// TwinCAT 3 PLC project TwinCAT_OpenFramework_Devices_IO
// Title: TwinCAT Open Framework Devices IO
// Company: Oleksandr Tiutyk FOP
// Author: Oleksandr Tiutyk
// ProjectVersion: 1.0.13.0
// Description: IO devices implementation
// ProgramVersion: 3.1.4026.28
// libraries:
//   Tc2_System, * (Beckhoff Automation GmbH)
//   [TwinCAT Open Framework Automation], * (Oleksandr Tiutyk FOP)
//   [TwinCAT Open Framework Core], * (Oleksandr Tiutyk FOP)
//   [TwinCAT Open Framework IO Models], * (Oleksandr Tiutyk FOP)
// project tree:
//   Analog/Inputs/ IAnalogInputStatusProvider.TcIO, IReadOnlyAnalogInput.TcIO, AnalogInput.TcPOU (not stored), ANALOG_INPUT_STATUS.TcPOU, IAnalogInput.TcIO
//   Analog/Outputs/ IReadOnlyAnalogOutput.TcIO, AnalogOutput.TcPOU, IAnalogOutput.TcIO
//   Analog/ RawAnalogValues.TcPOU, RAW_ANALOG_VALUE.TcDUT, IAnalogValueConverter.TcIO, RAW_ANALOG_VALUE_TYPE.TcDUT
//   Analog/StandardConverters/ DirectAnalogValueConverter.TcPOU
//   Analog/StandardConverters/Range/ AbstractRangeAnalogValueConverter.TcPOU, DynamicRangeAnalogValueConverter.TcPOU, StaticRangeAnalogValueConverter.TcPOU
//   / CONTACT_TYPE.TcDUT
//   Digital/Input/ DigitalInput.TcPOU, IDigitalInput.TcIO, IReadOnlyDigitalInput.TcIO
//   Digital/Output/ DigitalOutput.TcPOU, IReadOnlyDigitalOutput.TcIO, IDigitalOutput.TcIO
//   Internal/ CurrentNamespace.TcPOU, NamespaceExtractor.TcPOU
//   Version/ Global_Version.TcGVL
// (motion and I/O tree: see PLC project twincat_openframework_core)
// real-time tasks:
//   TASK PlcTask: cycle T#10ms, priority 20, ADS port 350
//   TASK TestTask: cycle T#10ms, priority 1, ADS port 351
//   TASK RunnerTestTask: cycle T#10ms, priority 2, ADS port 354
//   TASK HowToTask: cycle T#10ms, priority 22, ADS port 353
// variable links:

// ---- Analog/RAW_ANALOG_VALUE.TcDUT
(*
SPDX-FileCopyrightText: Â© 2026 Oleksandr Tiutyk <trofimich@gmail.com>
SPDX-License-Identifier: MIT
License: https://opensource.org/license/mit
*)

(*!
<summary>4-byte union representing raw analog process data.</summary>
<description>
Allows interpreting a 4-byte raw analog signal as signed 16-bit integer, signed 32-bit integer,
or single-precision 32-bit floating point.
</description>
*)

TYPE RAW_ANALOG_VALUE :
UNION
	Int16 : INT;
	Int32 : DINT;
	Real32 : REAL; 
END_UNION
END_TYPE

// ---- Analog/RAW_ANALOG_VALUE_TYPE.TcDUT
(*
SPDX-FileCopyrightText: Â© 2026 Oleksandr Tiutyk <trofimich@gmail.com>
SPDX-License-Identifier: MIT
License: https://opensource.org/license/mit
*)

(*!
<summary>Identifies underlying data type of a raw ADC or DAC analog signal.</summary>
<description>
Specifies whether the raw process data is interpreted as signed 16-bit integer, signed 32-bit integer,
or 32-bit single-precision floating point.
</description>
*)

{attribute 'qualified_only'}
{attribute 'strict'}
{attribute 'to_string'}
TYPE RAW_ANALOG_VALUE_TYPE :
(
	INT16,
	INT32,
	REAL32 
);
END_TYPE

// ---- CONTACT_TYPE.TcDUT
(*
SPDX-FileCopyrightText: © 2026 Oleksandr Tiutyk <trofimich@gmail.com>
SPDX-License-Identifier: MIT
License: https://opensource.org/license/mit
*)

(*!
<summary>Defines electrical contact type for digital input and output signals.</summary>
<description>
Determines whether the physical signal state is inverted when mapped to the logical component Value.
NORMALLY_OPEN: logical TRUE matches physical TRUE. NORMALLY_CLOSED: logical TRUE matches physical FALSE
(inverted).
</description>
*)

{attribute 'qualified_only'}
{attribute 'strict'}
{attribute 'to_string'}
TYPE CONTACT_TYPE :
(
	NORMALLY_OPEN := 0,
	NORMALLY_CLOSED := 1
);
END_TYPE

// ---- Version/Global_Version.TcGVL
{attribute 'TcGenerated'}
{attribute 'no-analysis'}
{attribute 'linkalways'}
// This function has been automatically generated from the project information.
VAR_GLOBAL CONSTANT
	{attribute 'const_non_replaced'}
	stLibVersion_TwinCAT_Open_Framework_Devices_IO : ST_LibVersion := (iMajor := 1, iMinor := 0, iBuild := 13, iRevision := 0, nFlags := 0, sVersion := '1.0.13.0');
END_VAR

// ---- Analog/Inputs/IAnalogInputStatusProvider.TcIO
(*
SPDX-FileCopyrightText: © 2026 Oleksandr Tiutyk <trofimich@gmail.com>
SPDX-License-Identifier: MIT
License: https://opensource.org/license/mit
*)

(*!
<summary>Exposes the sampled analog input channel status by value.</summary>
<description>
A consumer of IReadOnlyAnalogInput can query this separate interface when the input supports snapshots.
</description>
*)
INTERFACE IAnalogInputStatusProvider EXTENDS TOF_Core.IObject

(*!
<summary>Gets a copy of the channel status word sampled by ProcessInput().</summary>
<description>
Returns zero before the first sample and after processing input without a status binding. Read this value
from the input's owner task. Callers can freely modify their local copy.
</description>
*)
{attribute 'monitoring' := 'call'}
PROPERTY StatusWord : WORD
GET
END_GET
END_PROPERTY

END_INTERFACE

// ---- Analog/Inputs/IReadOnlyAnalogInput.TcIO
(*
SPDX-FileCopyrightText: Â© 2026 Oleksandr Tiutyk <trofimich@gmail.com>
SPDX-License-Identifier: MIT
License: https://opensource.org/license/mit
*)

(*!
<summary>Read-only contract for an analog input component.</summary>
<description>
Provides access to engineering value, raw converter, raw ADC value, legacy decoded status, and I/O binding.
Query IAnalogInputStatusProvider for the sampled status word by value when the implementation supports it.
</description>
*)
INTERFACE IReadOnlyAnalogInput EXTENDS TOF_Automation.IInputLeafAutomationComponent,
	TOF_Core.IIOBindable

(*!
<summary>Gets the assigned analog value converter.</summary>
*)
{attribute 'monitoring' := 'call'}
PROPERTY Converter : IAnalogValueConverter
GET
END_GET
END_PROPERTY

(*!
<summary>Gets current raw hardware ADC value cast to LREAL.</summary>
*)
{attribute 'monitoring' := 'call'}
PROPERTY RawValue : LREAL
GET
END_GET
END_PROPERTY

(*!
<summary>Gets the raw analog data representation type.</summary>
*)
{attribute 'monitoring' := 'call'}
PROPERTY RawValueType : RAW_ANALOG_VALUE_TYPE
GET
END_GET
END_PROPERTY

(*!
<summary>Gets a borrowed reference to the legacy decoded channel status.</summary>
<description>
The reference requires a live input and exposes a mutable decoder. AnalogInput refreshes this view in
ProcessInput() and uses a separate sampled word for diagnostics. Use IAnalogInputStatusProvider.StatusWord
when the implementation supports reading the sampled status by value.
</description>
*)
{attribute 'monitoring' := 'call'}
PROPERTY Status : REFERENCE TO ANALOG_INPUT_STATUS
GET
END_GET
END_PROPERTY

(*!
<summary>Gets current scaled engineering unit value.</summary>
*)
{attribute 'monitoring' := 'call'}
PROPERTY Value : LREAL
GET
END_GET
END_PROPERTY

END_INTERFACE

// ---- Analog/Outputs/IReadOnlyAnalogOutput.TcIO
(*
SPDX-FileCopyrightText: Â© 2026 Oleksandr Tiutyk <trofimich@gmail.com>
SPDX-License-Identifier: MIT
License: https://opensource.org/license/mit
*)

(*!
<summary>Read-only contract for an analog output automation component.</summary>
<description>
Provides access to engineering output value, assigned converter and raw representation.
</description>
*)

INTERFACE IReadOnlyAnalogOutput EXTENDS TOF_Automation.IOutputLeafAutomationComponent

(*!
<summary>Gets the assigned analog value converter.</summary>
*)
{attribute 'monitoring' := 'call'}
PROPERTY Converter : IAnalogValueConverter
GET
END_GET
END_PROPERTY

(*!
<summary>Gets current raw hardware DAC value cast to LREAL.</summary>
*)
{attribute 'monitoring' := 'call'}
PROPERTY RawValue : LREAL
GET
END_GET
END_PROPERTY

(*!
<summary>Gets the raw analog data representation type.</summary>
*)
{attribute 'monitoring' := 'call'}
PROPERTY RawValueType : RAW_ANALOG_VALUE_TYPE
GET
END_GET
END_PROPERTY

(*!
<summary>Gets current scaled engineering unit output value.</summary>
*)
{attribute 'monitoring' := 'call'}
PROPERTY Value : LREAL
GET
END_GET
END_PROPERTY

END_INTERFACE

// ---- Analog/IAnalogValueConverter.TcIO
(*
SPDX-FileCopyrightText: Â© 2026 Oleksandr Tiutyk <trofimich@gmail.com>
SPDX-License-Identifier: MIT
License: https://opensource.org/license/mit
*)

(*!
<summary>Contract for analog signal scaling and engineering unit conversion.</summary>
<description>
Converts raw ADC/DAC values to and from engineering unit LREAL representations.
</description>
*)

INTERFACE IAnalogValueConverter EXTENDS TOF_Core.IObject

(*!
<summary>Converts an engineering unit value to raw hardware representation.</summary>
<param name="analogValue">Engineering unit analog value.</param>
<param name="rawValueType">Target raw data representation.</param>
*)
METHOD ConvertAnalogValueToRawValue : RAW_ANALOG_VALUE
VAR_INPUT
	analogValue : LREAL;
	rawValueType : RAW_ANALOG_VALUE_TYPE;
END_VAR
END_METHOD

(*!
<summary>Converts raw hardware representation to an engineering unit value.</summary>
<param name="rawValue">Raw process value union.</param>
<param name="rawValueType">Source raw data representation.</param>
*)
METHOD ConvertRawValueToAnalogValue : LREAL
VAR_INPUT
	rawValue : RAW_ANALOG_VALUE;
	rawValueType : RAW_ANALOG_VALUE_TYPE;
END_VAR
END_METHOD

END_INTERFACE

// ---- Analog/Inputs/IAnalogInput.TcIO
(*
SPDX-FileCopyrightText: Â© 2026 Oleksandr Tiutyk <trofimich@gmail.com>
SPDX-License-Identifier: MIT
License: https://opensource.org/license/mit
*)

(*!
<summary>Contract for an analog input component with channel and scalar binding capabilities.</summary>
<description>
Extends IReadOnlyAnalogInput with hardware binding methods for compound Beckhoff channels
or standalone scalar input variables.
</description>
*)
INTERFACE IAnalogInput EXTENDS IReadOnlyAnalogInput

(*!
<summary>Binds component to a 16-bit analog input channel process image structure.</summary>
<description>
Borrows the channel fields without modifying the process image. The caller keeps the channel alive while bound
and synchronizes rebinding with input processing. An invalid reference clears value and status bindings.
</description>
<param name="rawValues">Reference to channel process structure containing Status and INT Value.</param>
*)
METHOD BindToInt16IO
VAR_INPUT
	rawValues : REFERENCE TO TOF_IOModels.ANALOG_INPUT_INT_CHANNEL;
END_VAR
END_METHOD

(*!
<summary>Binds component directly to a 16-bit signed integer raw input value.</summary>
<param name="rawValue">Reference to raw INT input variable.</param>
*)
METHOD BindToInt16Value
VAR_INPUT
	rawValue : REFERENCE TO INT;
END_VAR
END_METHOD

(*!
<summary>Binds component to a 32-bit analog input channel process image structure.</summary>
<description>
Borrows the channel fields without modifying source data. The caller keeps storage alive while bound
and synchronizes rebinding with processing. An invalid reference clears value and status bindings.
The channel must use the status-plus-DINT PDO; no compact-layout or unit conversion is performed here.
</description>
<param name="rawValues">Reference to channel process structure containing Status and DINT Value.</param>
*)
METHOD BindToInt32IO
VAR_INPUT
	rawValues : REFERENCE TO TOF_IOModels.ANALOG_INPUT_DINT_CHANNEL;
END_VAR
END_METHOD

(*!
<summary>Binds component directly to a 32-bit signed integer raw input value.</summary>
<param name="rawValue">Reference to raw DINT input variable.</param>
*)
METHOD BindToInt32Value
VAR_INPUT
	rawValue : REFERENCE TO DINT;
END_VAR
END_METHOD

(*!
<summary>Binds component to a 32-bit float analog input channel process image structure.</summary>
<description>
Borrows the channel fields without modifying source data. The caller keeps storage alive while bound
and synchronizes rebinding with processing. An invalid reference clears value and status bindings.
The channel must use the status-plus-REAL PDO; no integer-layout or unit conversion is performed here.
</description>
<param name="rawValues">Reference to channel process structure containing Status and REAL Value.</param>
*)
METHOD BindToReal32IO
VAR_INPUT
	rawValues : REFERENCE TO TOF_IOModels.ANALOG_INPUT_REAL_CHANNEL;
END_VAR
END_METHOD

(*!
<summary>Binds component directly to a 32-bit single-precision float raw input value.</summary>
<param name="rawValue">Reference to raw REAL input variable.</param>
*)
METHOD BindToReal32Value
VAR_INPUT
	rawValue : REFERENCE TO REAL;
END_VAR
END_METHOD

END_INTERFACE

// ---- Analog/Outputs/IAnalogOutput.TcIO
(*
SPDX-FileCopyrightText: Â© 2026 Oleksandr Tiutyk <trofimich@gmail.com>
SPDX-License-Identifier: MIT
License: https://opensource.org/license/mit
*)

(*!
<summary>Configuration and control contract for an analog output component.</summary>
<description>
Extends IReadOnlyAnalogOutput with hardware IO binding methods and value mutator.
</description>
*)

INTERFACE IAnalogOutput EXTENDS IReadOnlyAnalogOutput

(*!
<summary>Binds component to a 16-bit signed integer output process image variable '%Q*'.</summary>
<param name="rawVariable">Reference to physical INT output variable.</param>
*)
METHOD BindToInt16IO
VAR_INPUT
	rawVariable : REFERENCE TO INT;
END_VAR
END_METHOD

(*!
<summary>Binds component to a 32-bit signed integer output process image variable '%Q*'.</summary>
<param name="rawVariable">Reference to physical DINT output variable.</param>
*)
METHOD BindToInt32IO
VAR_INPUT
	rawVariable : REFERENCE TO DINT;
END_VAR
END_METHOD

(*!
<summary>Binds component to a 32-bit float output process image variable '%Q*'.</summary>
<param name="rawVariable">Reference to physical REAL output variable.</param>
*)
METHOD BindToReal32IO
VAR_INPUT
	rawVariable : REFERENCE TO REAL;
END_VAR
END_METHOD

(*!
<summary>Gets or sets engineering unit value to output.</summary>
*)
{attribute 'monitoring' := 'call'}
PROPERTY Value : LREAL
GET
END_GET
SET
END_SET
END_PROPERTY

END_INTERFACE

// ---- Digital/Input/IDigitalInput.TcIO
(*
SPDX-FileCopyrightText: Â© 2026 Oleksandr Tiutyk <trofimich@gmail.com>
SPDX-License-Identifier: MIT
License: https://opensource.org/license/mit
*)

(*!
<summary>Configuration and binding contract for a digital input component.</summary>
<description>
Extends IReadOnlyDigitalInput with hardware IO mapping and contact type mutator.
</description>
*)

INTERFACE IDigitalInput EXTENDS IReadOnlyDigitalInput

(*!
<summary>Binds the component to a raw boolean process image variable.</summary>
<param name="rawValue">Reference to physical boolean input variable '%I*'.</param>
*)
METHOD BindToIO
VAR_INPUT
	rawValue : REFERENCE TO BOOL;
END_VAR
END_METHOD

(*!
<summary>Gets or sets electrical contact configuration.</summary>
*)
{attribute 'monitoring' := 'call'}
PROPERTY ContactType : CONTACT_TYPE
GET
END_GET
SET
END_SET
END_PROPERTY

END_INTERFACE

// ---- Digital/Input/IReadOnlyDigitalInput.TcIO
(*
SPDX-FileCopyrightText: Â© 2026 Oleksandr Tiutyk <trofimich@gmail.com>
SPDX-License-Identifier: MIT
License: https://opensource.org/license/mit
*)

(*!
<summary>Read-only contract for a digital input automation component.</summary>
<description>
Provides access to logical boolean state, change detection and electrical contact configuration.
</description>
*)

INTERFACE IReadOnlyDigitalInput EXTENDS TOF_Automation.IInputLeafAutomationComponent

(*!
<summary>Indicates whether the logical Value has changed compared to the previous cycle.</summary>
*)
{attribute 'monitoring' := 'call'}
PROPERTY Changed : BOOL
GET
END_GET
END_PROPERTY

(*!
<summary>Gets electrical contact configuration (normally open or normally closed).</summary>
*)
{attribute 'monitoring' := 'call'}
PROPERTY ContactType : CONTACT_TYPE
GET
END_GET
END_PROPERTY

(*!
<summary>Gets current evaluated logical state of the input signal.</summary>
*)
{attribute 'monitoring' := 'call'}
PROPERTY Value : BOOL
GET
END_GET
END_PROPERTY

END_INTERFACE

// ---- Digital/Output/IReadOnlyDigitalOutput.TcIO
(*
SPDX-FileCopyrightText: Â© 2026 Oleksandr Tiutyk <trofimich@gmail.com>
SPDX-License-Identifier: MIT
License: https://opensource.org/license/mit
*)

(*!
<summary>Read-only contract for a digital output automation component.</summary>
<description>
Provides access to logical boolean output state, change detection and electrical contact configuration.
</description>
*)

INTERFACE IReadOnlyDigitalOutput EXTENDS TOF_Automation.IOutputLeafAutomationComponent

(*!
<summary>Indicates whether the current logical command differs from the last processed command.</summary>
<description>
ProcessOutput() acknowledges the current command even without an I/O binding.
</description>
*)
{attribute 'monitoring' := 'call'}
PROPERTY Changed : BOOL
GET
END_GET
END_PROPERTY

(*!
<summary>Gets electrical contact configuration.</summary>
*)
{attribute 'monitoring' := 'call'}
PROPERTY ContactType : CONTACT_TYPE
GET
END_GET
END_PROPERTY

(*!
<summary>Gets current evaluated logical state of the output signal.</summary>
*)
{attribute 'monitoring' := 'call'}
PROPERTY Value : BOOL
GET
END_GET
END_PROPERTY

END_INTERFACE

// ---- Digital/Output/IDigitalOutput.TcIO
(*
SPDX-FileCopyrightText: Â© 2026 Oleksandr Tiutyk <trofimich@gmail.com>
SPDX-License-Identifier: MIT
License: https://opensource.org/license/mit
*)

(*!
<summary>Configuration and control contract for a digital output component.</summary>
<description>
Extends IReadOnlyDigitalOutput with hardware IO mapping, contact configuration and state setter.
</description>
*)

INTERFACE IDigitalOutput EXTENDS IReadOnlyDigitalOutput

(*!
<summary>Binds component to a raw boolean process image output variable.</summary>
<param name="rawValue">Reference to physical boolean output variable '%Q*'.</param>
*)
METHOD BindToIO
VAR_INPUT
	rawValue : REFERENCE TO BOOL;
END_VAR
END_METHOD

(*!
<summary>Gets or sets electrical contact configuration.</summary>
*)
{attribute 'monitoring' := 'call'}
PROPERTY ContactType : CONTACT_TYPE
GET
END_GET
SET
END_SET
END_PROPERTY

(*!
<summary>Gets or sets logical state to write to the digital output.</summary>
*)
{attribute 'monitoring' := 'call'}
PROPERTY Value : BOOL
GET
END_GET
SET
END_SET
END_PROPERTY

END_INTERFACE

// ---- Analog/RawAnalogValues.TcPOU
(*
SPDX-FileCopyrightText: Â© 2026 Oleksandr Tiutyk <trofimich@gmail.com>
SPDX-License-Identifier: MIT
License: https://opensource.org/license/mit
*)

(*!
<summary>Utility program providing factory methods to construct RAW_ANALOG_VALUE unions.</summary>
<description>
Ensures that unused bytes of the 4-byte union are zero-initialized when constructing from 16-bit values.
</description>
*)

{attribute 'no_explicit_call' := 'do not call this POU directly'}
PROGRAM RawAnalogValues
VAR
	{attribute 'hide'} 
	_ClassName : STRING := __POUNAME();
END_VAR

(*!
<summary>Gets the class name of the program.</summary>
*)
{attribute 'monitoring' := 'call'}
PROPERTY ClassName : REFERENCE TO STRING
GET
ClassName REF= _ClassName;
END_GET
END_PROPERTY

(*!
<summary>Creates a RAW_ANALOG_VALUE union from a 16-bit signed integer.</summary>
<description>Zeroes upper bytes of the 4-byte union before assigning the 16-bit value.</description>
<param name="value">16-bit signed integer value.</param>
*)
METHOD FromInt16 : RAW_ANALOG_VALUE
VAR_INPUT
	value : INT;
END_VAR
FromInt16.Int32 := 0;
FromInt16.Int16 := value;
END_METHOD

(*!
<summary>Creates a RAW_ANALOG_VALUE union from a 32-bit signed integer.</summary>
<param name="value">32-bit signed integer value.</param>
*)
METHOD FromInt32 : RAW_ANALOG_VALUE
VAR_INPUT
	value : DINT;
END_VAR
FromInt32.Int32 := value;
END_METHOD

(*!
<summary>Creates a RAW_ANALOG_VALUE union from a 32-bit single-precision float.</summary>
<param name="value">32-bit float value.</param>
*)
METHOD FromReal32 : RAW_ANALOG_VALUE
VAR_INPUT
	value : REAL;
END_VAR
FromReal32.Real32 := value;
END_METHOD

(*!
<summary>Gets the namespace name of the program.</summary>
*)
{attribute 'monitoring' := 'call'}
PROPERTY NamespaceName : REFERENCE TO STRING
GET
NamespaceName REF= CurrentNamespace.Name;
END_GET
END_PROPERTY

END_PROGRAM

// ---- Internal/CurrentNamespace.TcPOU
(*
SPDX-FileCopyrightText: Â© 2026 Oleksandr Tiutyk <trofimich@gmail.com>
SPDX-License-Identifier: MIT
License: https://opensource.org/license/mit
*)

(*!
<summary>Internal program providing library namespace extraction.</summary>
*)

{attribute 'no_explicit_call' := 'do not call this POU directly'}
PROGRAM INTERNAL CurrentNamespace
VAR
	{attribute 'hide'} 
	_NamespaceExtractor : NamespaceExtractor;
END_VAR

(*!
<summary>Gets the effective namespace of this library.</summary>
*)
{attribute 'monitoring' := 'call'}
PROPERTY Name : REFERENCE TO STRING
GET
Name REF= _NamespaceExtractor.CurrentNamespace;
END_GET
END_PROPERTY

END_PROGRAM

// ---- Internal/NamespaceExtractor.TcPOU
(*
SPDX-FileCopyrightText: Â© 2026 Oleksandr Tiutyk <trofimich@gmail.com>
SPDX-License-Identifier: MIT
License: https://opensource.org/license/mit
*)

(*!
<summary>Internal function block that extracts the library namespace via init_namespace attribute.</summary>
*)

FUNCTION_BLOCK INTERNAL NamespaceExtractor
VAR_OUTPUT
	{attribute 'init_namespace'} 
	CurrentNamespace : STRING; 	
END_VAR

END_FUNCTION_BLOCK

// ---- Analog/Inputs/ANALOG_INPUT_STATUS.TcPOU
(*
SPDX-FileCopyrightText: Â© 2026 Oleksandr Tiutyk <trofimich@gmail.com>
SPDX-License-Identifier: MIT
License: https://opensource.org/license/mit
*)

(*!
<summary>Encapsulates and decodes Beckhoff 16-bit EtherCAT analog input status word.</summary>
<description>
Provides decoded boolean properties for Underrange (bit 0), Overrange (bit 1), Limit 1 (bits 2..3),
Limit 2 (bits 4..5), Error (bit 6), TxPDO State (bit 14), and TxPDO Toggle (bit 15).
</description>
*)

FUNCTION_BLOCK ANALOG_INPUT_STATUS
VAR
	_Status : WORD;
END_VAR

(*!
<summary>Bit 6: General measurement or hardware error flag.</summary>
*)
{attribute 'monitoring' := 'call'}
PROPERTY FINAL Error : BOOL
GET
Error := _Status.6;
END_GET
END_PROPERTY

(*!
<summary>Bit 1: Upper limit of nominal measuring range exceeded.</summary>
*)
{attribute 'monitoring' := 'call'}
PROPERTY FINAL Overrange : BOOL
GET
Overrange := _Status.1;
END_GET
END_PROPERTY

(*!
<summary>Updates internal raw 16-bit status word.</summary>
<param name="status">Raw 16-bit EtherCAT channel status word.</param>
*)
METHOD SetStatus
VAR_INPUT
	status : WORD;
END_VAR
_Status := status;
END_METHOD

(*!
<summary>Bit 14: TxPDO data validity (0: valid, 1: invalid / bus error).</summary>
*)
{attribute 'monitoring' := 'call'}
PROPERTY FINAL TxPDOState : BOOL
GET
TxPDOState := _Status.14;
END_GET
END_PROPERTY

(*!
<summary>Bit 15: TxPDO communication toggle bit.</summary>
*)
{attribute 'monitoring' := 'call'}
PROPERTY FINAL TxPDOToggle : BOOL
GET
TxPDOToggle := _Status.15;
END_GET
END_PROPERTY

(*!
<summary>Bit 0: Lower limit of calibrated measuring range fallen below.</summary>
*)
{attribute 'monitoring' := 'call'}
PROPERTY FINAL Underrange : BOOL
GET
Underrange := _Status.0;
END_GET
END_PROPERTY

(*!
<summary>Bit 3: Input value is greater than or equal to Limit 1 threshold.</summary>
*)
{attribute 'monitoring' := 'call'}
PROPERTY FINAL ValueBiggerOrEqualLimit1 : BOOL
GET
ValueBiggerOrEqualLimit1 := _Status.3;
END_GET
END_PROPERTY

(*!
<summary>Bit 5: Input value is greater than or equal to Limit 2 threshold.</summary>
*)
{attribute 'monitoring' := 'call'}
PROPERTY FINAL ValueBiggerOrEqualLimit2 : BOOL
GET
ValueBiggerOrEqualLimit2 := _Status.5;
END_GET
END_PROPERTY

(*!
<summary>Bit 2: Input value is smaller than or equal to Limit 1 threshold.</summary>
*)
{attribute 'monitoring' := 'call'}
PROPERTY FINAL ValueSmallerOrEqualLimit1 : BOOL
GET
ValueSmallerOrEqualLimit1 := _Status.2;
END_GET
END_PROPERTY

(*!
<summary>Bit 4: Input value is smaller than or equal to Limit 2 threshold.</summary>
*)
{attribute 'monitoring' := 'call'}
PROPERTY FINAL ValueSmallerOrEqualLimit2 : BOOL
GET
ValueSmallerOrEqualLimit2 := _Status.4;
END_GET
END_PROPERTY

END_FUNCTION_BLOCK

// ---- Analog/Outputs/AnalogOutput.TcPOU
(*
SPDX-FileCopyrightText: Â© 2026 Oleksandr Tiutyk <trofimich@gmail.com>
SPDX-License-Identifier: MIT
License: https://opensource.org/license/mit
*)

(*!
<summary>Analog output automation component converting engineering values into raw DAC signals.</summary>
<description>
Scales engineering unit values using an assigned IAnalogValueConverter and writes raw data to hardware outputs.
Successful initialization requires a parent automation component.
</description>
*)

FUNCTION_BLOCK AnalogOutput EXTENDS TOF_Automation.OutputLeafAutomationComponent
	IMPLEMENTS IAnalogOutput, TOF_Core.IIOBindable
VAR_STAT
	{attribute 'hide'} 
	_ClassName : STRING := __POUNAME();
END_VAR
VAR	
	{attribute 'hide'} 
	_RawValueType : RAW_ANALOG_VALUE_TYPE;

	{attribute 'hide'} 
	_Converter : IAnalogValueConverter;

	_CurrentValue : LREAL;
	_PreviousValue : LREAL;
	
	_RawInt16Value : REFERENCE TO INT;
	_RawInt32Value : REFERENCE TO DINT;
	_RawReal32Value : REFERENCE TO REAL; 
END_VAR

(*!
<summary>Binds component to a 16-bit signed integer output process image variable '%Q*'.</summary>
<param name="rawVariable">Reference to physical INT output variable.</param>
*)
METHOD BindToInt16IO
VAR_INPUT
	rawVariable : REFERENCE TO INT;
END_VAR
_RawValueType := RAW_ANALOG_VALUE_TYPE.INT16;

_RawInt16Value REF= rawVariable;
_RawInt32Value REF= 0;
_RawReal32Value REF= 0;
END_METHOD

(*!
<summary>Binds component to a 32-bit signed integer output process image variable '%Q*'.</summary>
<param name="rawVariable">Reference to physical DINT output variable.</param>
*)
METHOD BindToInt32IO
VAR_INPUT
	rawVariable : REFERENCE TO DINT;
END_VAR
_RawValueType := RAW_ANALOG_VALUE_TYPE.INT32;

_RawInt16Value REF= 0;
_RawInt32Value REF= rawVariable;
_RawReal32Value REF= 0;
END_METHOD

(*!
<summary>Binds component to a 32-bit float output process image variable '%Q*'.</summary>
<param name="rawVariable">Reference to physical REAL output variable.</param>
*)
METHOD BindToReal32IO
VAR_INPUT
	rawVariable : REFERENCE TO REAL;
END_VAR
_RawValueType := RAW_ANALOG_VALUE_TYPE.REAL32;

_RawInt16Value REF= 0;
_RawInt32Value REF= 0;
_RawReal32Value REF= rawVariable;
END_METHOD

(*!
<summary>Gets whether the component raw value is bound to a valid physical IO variable.</summary>
*)
{attribute 'monitoring' := 'call'}
PROPERTY FINAL BoundToIO : BOOL
GET
CASE _RawValueType OF
	RAW_ANALOG_VALUE_TYPE.INT16:
		BoundToIO := __ISVALIDREF(_RawInt16Value);
	
	RAW_ANALOG_VALUE_TYPE.INT32:
		BoundToIO := __ISVALIDREF(_RawInt32Value);
	
	RAW_ANALOG_VALUE_TYPE.REAL32:
		BoundToIO := __ISVALIDREF(_RawReal32Value);
END_CASE
END_GET
END_PROPERTY

(*!
<summary>Gets the class name of the component.</summary>
*)
{attribute 'monitoring' := 'call'}
PROPERTY ClassName : REFERENCE TO STRING
GET
ClassName REF= _ClassName;
END_GET
END_PROPERTY

(*!
<summary>Gets the assigned analog value converter.</summary>
*)
{attribute 'monitoring' := 'call'}
PROPERTY FINAL Converter : IAnalogValueConverter
GET
Converter := _Converter;
END_GET
END_PROPERTY

(*!
<summary>Initializes component name, parent and converter dependency.</summary>
<param name="bInitRetains">TRUE: retain variables are initialized.</param>
<param name="bInCopyCode">TRUE: instance copied to copy code (online change).</param>
<param name="name">Component instance name.</param>
<param name="parent">Nonzero parent automation component required for successful Initialize().</param>
<param name="converter">Mandatory analog value converter dependency.</param>
*)
METHOD FB_init : BOOL
VAR_INPUT
	bInitRetains : BOOL; // TRUE: the retain variables are initialized (reset warm / reset cold)
	bInCopyCode : BOOL;  // TRUE: the instance will be copied to the copy code afterward (online change)
	name : WSTRING;
	parent : TOF_Automation.IParentAutomationComponent;
	converter : IAnalogValueConverter;
END_VAR
IF NOT bInCopyCode THEN
	_Converter := converter;
END_IF
END_METHOD

(*!
<summary>Gets the namespace name of the component.</summary>
*)
{attribute 'monitoring' := 'call'}
PROPERTY NamespaceName : REFERENCE TO STRING
GET
NamespaceName REF= CurrentNamespace.Name;
END_GET
END_PROPERTY

(*!
<summary>Validates that mandatory converter dependency is configured.</summary>
*)
METHOD PROTECTED OnInitializing : BOOL
IF _Converter = 0 THEN
	TOF_Core.Exceptions.ThrowClassInitialization(
		sourceNamespaceName := NamespaceName,
		sourceClassName := ClassName,
		sourcePOUName := __POUNAME(),
		sourcePosition := __POSITION(),
		errorMessage := "converter not specified"
	);
END_IF

OnInitializing := TRUE;
END_METHOD

(*!
<summary>Scales engineering value to raw DAC signal and writes to bound hardware output.</summary>
*)
METHOD PROTECTED OnProcessOutput
setRawValueByUnion(
	_Converter.ConvertAnalogValueToRawValue(
		analogValue := _CurrentValue,
		rawValueType := _RawValueType
	)
);

_PreviousValue := _CurrentValue;
END_METHOD

(*!
<summary>Gets current raw hardware DAC value cast to LREAL.</summary>
*)
{attribute 'monitoring' := 'call'}
PROPERTY FINAL RawValue : LREAL
GET
CASE _RawValueType OF
	RAW_ANALOG_VALUE_TYPE.INT16:
		RawValue := SEL(__ISVALIDREF(_RawInt16Value), 0, TO_LREAL(_RawInt16Value));
	
	RAW_ANALOG_VALUE_TYPE.INT32:
		RawValue := SEL(__ISVALIDREF(_RawInt32Value), 0, TO_LREAL(_RawInt32Value));
	
	RAW_ANALOG_VALUE_TYPE.REAL32:
		RawValue := SEL(__ISVALIDREF(_RawReal32Value), 0, TO_LREAL(_RawReal32Value));
END_CASE
END_GET
END_PROPERTY

(*!
<summary>Gets the raw analog data representation type.</summary>
*)
{attribute 'monitoring' := 'call'}
PROPERTY FINAL RawValueType : RAW_ANALOG_VALUE_TYPE
GET
RawValueType := _RawValueType;
END_GET
END_PROPERTY

(*!
<summary>Gets the memory size of the instance.</summary>
*)
{attribute 'monitoring' := 'call'}
PROPERTY SelfSize : ULINT
GET
SelfSize := XSIZEOF(THIS^);
END_GET
END_PROPERTY

METHOD PRIVATE setRawValueByUnion
VAR_INPUT
	rawValueUnion : RAW_ANALOG_VALUE;
END_VAR
CASE _RawValueType OF
	RAW_ANALOG_VALUE_TYPE.INT16:
		IF __ISVALIDREF(_RawInt16Value) THEN
			_RawInt16Value := rawValueUnion.Int16; 
		END_IF
	
	RAW_ANALOG_VALUE_TYPE.INT32:
		IF __ISVALIDREF(_RawInt32Value) THEN
			_RawInt32Value := rawValueUnion.Int32; 
		END_IF
	
	RAW_ANALOG_VALUE_TYPE.REAL32:
		IF __ISVALIDREF(_RawReal32Value) THEN
			_RawReal32Value := rawValueUnion.Real32; 
		END_IF
END_CASE
END_METHOD

(*!
<summary>Gets or sets engineering unit value to output.</summary>
*)
{attribute 'monitoring' := 'call'}
PROPERTY Value : LREAL
GET
Value := _CurrentValue;
END_GET
SET
_CurrentValue := Value;
END_SET
END_PROPERTY

END_FUNCTION_BLOCK

// ---- Analog/StandardConverters/DirectAnalogValueConverter.TcPOU
(*
SPDX-FileCopyrightText: Â© 2026 Oleksandr Tiutyk <trofimich@gmail.com>
SPDX-License-Identifier: MIT
License: https://opensource.org/license/mit
*)

(*!
<summary>Performs direct 1:1 pass-through conversion between raw and engineering analog values.</summary>
<description>
Casts between numeric types without range scaling or boundary clamping.
</description>
*)

{attribute 'no_explicit_call' := 'do not call this function block directly'}
FUNCTION_BLOCK DirectAnalogValueConverter EXTENDS TOF_Core.Object IMPLEMENTS IAnalogValueConverter
VAR_STAT
	{attribute 'hide'} 
	_ClassName : STRING := __POUNAME();
END_VAR

(*!
<summary>Gets the class name of the converter.</summary>
*)
{attribute 'monitoring' := 'call'}
PROPERTY ClassName : REFERENCE TO STRING
GET
ClassName REF= _ClassName;
END_GET
END_PROPERTY

(*!
<summary>Directly converts an engineering unit value to raw hardware representation.</summary>
<param name="analogValue">Engineering unit analog value.</param>
<param name="rawValueType">Target raw data representation.</param>
*)
METHOD ConvertAnalogValueToRawValue : RAW_ANALOG_VALUE
VAR_INPUT
	analogValue	: LREAL;
	rawValueType : RAW_ANALOG_VALUE_TYPE;
END_VAR
ConvertAnalogValueToRawValue.Int32 := 0;

CASE rawValueType OF
	RAW_ANALOG_VALUE_TYPE.INT16:
		ConvertAnalogValueToRawValue.Int16 := TO_INT(analogValue);
	
	RAW_ANALOG_VALUE_TYPE.INT32:
		ConvertAnalogValueToRawValue.Int32 := TO_DINT(analogValue);
	
	RAW_ANALOG_VALUE_TYPE.REAL32:
		ConvertAnalogValueToRawValue.Real32 := TO_REAL(analogValue);
	
	ELSE
		RETURN;
END_CASE
END_METHOD

(*!
<summary>Directly converts a raw hardware representation to an engineering unit value.</summary>
<param name="rawValue">Raw process value union.</param>
<param name="rawValueType">Source raw data representation.</param>
*)
METHOD ConvertRawValueToAnalogValue : LREAL
VAR_INPUT
	rawValue : RAW_ANALOG_VALUE;
	rawValueType : RAW_ANALOG_VALUE_TYPE;
END_VAR
CASE rawValueType OF
	RAW_ANALOG_VALUE_TYPE.INT16:
		ConvertRawValueToAnalogValue := TO_LREAL(rawValue.Int16);
	
	RAW_ANALOG_VALUE_TYPE.INT32:
		ConvertRawValueToAnalogValue := TO_LREAL(rawValue.Int32);
	
	RAW_ANALOG_VALUE_TYPE.REAL32:
		ConvertRawValueToAnalogValue := TO_LREAL(rawValue.Real32);
	
	ELSE
		ConvertRawValueToAnalogValue := 0;
END_CASE
END_METHOD

(*!
<summary>Gets the namespace name of the converter.</summary>
*)
{attribute 'monitoring' := 'call'}
PROPERTY NamespaceName : REFERENCE TO STRING
GET
NamespaceName REF= CurrentNamespace.Name;
END_GET
END_PROPERTY

(*!
<summary>Gets the memory size of the instance.</summary>
*)
{attribute 'monitoring' := 'call'}
PROPERTY SelfSize : ULINT
GET
SelfSize := XSIZEOF(THIS^);
END_GET
END_PROPERTY

END_FUNCTION_BLOCK

// ---- Analog/StandardConverters/Range/AbstractRangeAnalogValueConverter.TcPOU
(*
SPDX-FileCopyrightText: Â© 2026 Oleksandr Tiutyk <trofimich@gmail.com>
SPDX-License-Identifier: MIT
License: https://opensource.org/license/mit
*)

(*!
<summary>Base converter providing linear interpolation and boundary clamping
between raw and engineering values.</summary>
<description>
Maps an input value proportionally between configured minimum and maximum limits.
Clamps values outside range to boundary limits and defends against division by zero.
For a range with distinct engineering limits and equal raw limits, output conversion returns the common raw limit.
</description>
*)

{attribute 'no_explicit_call' := 'do not call this function block directly'}
FUNCTION_BLOCK ABSTRACT AbstractRangeAnalogValueConverter EXTENDS TOF_Core.Object IMPLEMENTS IAnalogValueConverter
VAR
	{attribute 'hide'} 
	_MinAnalogValue : REFERENCE TO LREAL;
	{attribute 'hide'} 
	_MaxAnalogValue : REFERENCE TO LREAL;
	{attribute 'hide'} 
	_MinRawValue : REFERENCE TO RAW_ANALOG_VALUE;
	{attribute 'hide'} 
	_MaxRawValue : REFERENCE TO RAW_ANALOG_VALUE;
END_VAR

(*!
<summary>Converts an engineering unit value to raw hardware representation with boundary clamping.</summary>
<description>
If the engineering limits differ and the raw limits are equal, returns the common limit in the requested
raw representation. An INT16 result has zeroed upper bytes.
</description>
<param name="analogValue">Engineering unit analog value.</param>
<param name="rawValueType">Target raw data representation.</param>
*)
METHOD ConvertAnalogValueToRawValue : RAW_ANALOG_VALUE
VAR_INPUT
	analogValue	: LREAL;
	rawValueType : RAW_ANALOG_VALUE_TYPE;
END_VAR
VAR
	formattedExceptionMessage : TOF_Core.ERROR_MESSAGE;

	minRawValueLReal : LREAL;
	maxRawValueLReal : LREAL;
	rawValueLReal : LREAL;
	
	exceptionCode : __SYSTEM.ExceptionCode;	
END_VAR
IF NOT __ISVALIDREF(_MinAnalogValue)
	OR_ELSE NOT __ISVALIDREF(_MaxAnalogValue)
	OR_ELSE NOT __ISVALIDREF(_MinRawValue)
	OR_ELSE NOT __ISVALIDREF(_MaxRawValue)
	OR_ELSE _MinAnalogValue = _MaxAnalogValue
THEN
	RETURN;
END_IF

IF _MaxAnalogValue > _MinAnalogValue THEN
	IF analogValue >= _MaxAnalogValue THEN
		analogValue := _MaxAnalogValue;
	ELSIF analogValue <= _MinAnalogValue THEN
		analogValue := _MinAnalogValue;
	END_IF
ELSIF _MaxAnalogValue < _MinAnalogValue THEN
	IF analogValue <= _MaxAnalogValue THEN
		analogValue := _MaxAnalogValue;
	ELSIF analogValue >= _MinAnalogValue THEN
		analogValue := _MinAnalogValue;
	END_IF
END_IF

CASE rawValueType OF
	RAW_ANALOG_VALUE_TYPE.INT16:
		minRawValueLReal := TO_LREAL(_MinRawValue.Int16);
		maxRawValueLReal := TO_LREAL(_MaxRawValue.Int16);

	RAW_ANALOG_VALUE_TYPE.INT32:
		minRawValueLReal := TO_LREAL(_MinRawValue.Int32);
		maxRawValueLReal := TO_LREAL(_MaxRawValue.Int32);

	RAW_ANALOG_VALUE_TYPE.REAL32:
		minRawValueLReal := TO_LREAL(_MinRawValue.Real32);
		maxRawValueLReal := TO_LREAL(_MaxRawValue.Real32);

	ELSE
		RETURN;
END_CASE

IF minRawValueLReal = maxRawValueLReal THEN
	CASE rawValueType OF
		RAW_ANALOG_VALUE_TYPE.INT16:
			ConvertAnalogValueToRawValue := RawAnalogValues.FromInt16(value := _MinRawValue.Int16);

		RAW_ANALOG_VALUE_TYPE.INT32:
			ConvertAnalogValueToRawValue := RawAnalogValues.FromInt32(value := _MinRawValue.Int32);

		RAW_ANALOG_VALUE_TYPE.REAL32:
			ConvertAnalogValueToRawValue := RawAnalogValues.FromReal32(value := _MinRawValue.Real32);
	END_CASE

	RETURN;
END_IF

__TRY
	rawValueLReal := (analogValue - _MinAnalogValue) / (_MaxAnalogValue - _MinAnalogValue)
		* (maxRawValueLReal - minRawValueLReal) + minRawValueLReal;
__CATCH(exceptionCode)
	formattedExceptionMessage := TOF_Core.WideStrings.Concat255(
		"Invalid analog to raw value conversion. Exception code: ",
		TO_WSTRING(exceptionCode)
	);

	TOF_Core.Exceptions.ThrowStandard(
		sourceNamespaceName := NamespaceName,
		sourceClassName := ClassName,
		sourcePOUName := __POUNAME(),
		sourcePosition := __POSITION(),
		message := formattedExceptionMessage
	);
__ENDTRY

ConvertAnalogValueToRawValue.Int32 := 0;

CASE rawValueType OF
	RAW_ANALOG_VALUE_TYPE.INT16:
		ConvertAnalogValueToRawValue.Int16 := TO_INT(rawValueLReal);

	RAW_ANALOG_VALUE_TYPE.INT32:
		ConvertAnalogValueToRawValue.Int32 := TO_DINT(rawValueLReal);

	RAW_ANALOG_VALUE_TYPE.REAL32:
		ConvertAnalogValueToRawValue.Real32 := TO_REAL(rawValueLReal);
END_CASE
END_METHOD

(*!
<summary>Converts raw hardware representation to an engineering unit value with boundary clamping.</summary>
<param name="rawValue">Raw process value union.</param>
<param name="rawValueType">Source raw data representation.</param>
*)
METHOD ConvertRawValueToAnalogValue : LREAL
VAR_INPUT
	rawValue : RAW_ANALOG_VALUE;
	rawValueType : RAW_ANALOG_VALUE_TYPE;
END_VAR
VAR
	formattedExceptionMessage : TOF_Core.ERROR_MESSAGE;

	rawValueLReal : LREAL;
	minRawValueLReal : LREAL;
	maxRawValueLReal : LREAL;

	exceptionCode : __SYSTEM.ExceptionCode;
END_VAR
IF NOT __ISVALIDREF(_MinAnalogValue)
	OR_ELSE NOT __ISVALIDREF(_MaxAnalogValue)
	OR_ELSE NOT __ISVALIDREF(_MinRawValue)
	OR_ELSE NOT __ISVALIDREF(_MaxRawValue)
	OR_ELSE _MinAnalogValue = _MaxAnalogValue
THEN
	RETURN;
END_IF

CASE rawValueType OF
	RAW_ANALOG_VALUE_TYPE.INT16:
		rawValueLReal := TO_LREAL(rawValue.Int16);
		minRawValueLReal := TO_LREAL(_MinRawValue.Int16);
		maxRawValueLReal := TO_LREAL(_MaxRawValue.Int16);

	RAW_ANALOG_VALUE_TYPE.INT32:
		rawValueLReal := TO_LREAL(rawValue.Int32);
		minRawValueLReal := TO_LREAL(_MinRawValue.Int32);
		maxRawValueLReal := TO_LREAL(_MaxRawValue.Int32);

	RAW_ANALOG_VALUE_TYPE.REAL32:
		rawValueLReal := TO_LREAL(rawValue.Real32);
		minRawValueLReal := TO_LREAL(_MinRawValue.Real32);
		maxRawValueLReal := TO_LREAL(_MaxRawValue.Real32);

	ELSE
		RETURN;
END_CASE

IF maxRawValueLReal > minRawValueLReal THEN
	IF rawValueLReal >= maxRawValueLReal THEN
		ConvertRawValueToAnalogValue := _MaxAnalogValue;
		RETURN;
	ELSIF rawValueLReal <= minRawValueLReal THEN
		ConvertRawValueToAnalogValue := _MinAnalogValue;
		RETURN;
	END_IF
ELSIF maxRawValueLReal < minRawValueLReal THEN
	IF rawValueLReal <= maxRawValueLReal THEN
		ConvertRawValueToAnalogValue := _MaxAnalogValue;
		RETURN;
	ELSIF rawValueLReal >= minRawValueLReal THEN
		ConvertRawValueToAnalogValue := _MinAnalogValue;
		RETURN;
	END_IF
ELSE
	ConvertRawValueToAnalogValue := _MinAnalogValue;
	RETURN;
END_IF

__TRY
	ConvertRawValueToAnalogValue := (rawValueLReal - minRawValueLReal) / (maxRawValueLReal - minRawValueLReal)
		* (_MaxAnalogValue - _MinAnalogValue) + _MinAnalogValue;
__CATCH(exceptionCode)
	formattedExceptionMessage := TOF_Core.WideStrings.Concat255(
		"Invalid raw to analog value conversion. Exception code: ",
		TO_WSTRING(exceptionCode)
	);

	TOF_Core.Exceptions.ThrowStandard(
		sourceNamespaceName := NamespaceName,
		sourceClassName := ClassName,
		sourcePOUName := __POUNAME(),
		sourcePosition := __POSITION(),
		message := formattedExceptionMessage
	);
__ENDTRY
END_METHOD

(*!
<summary>Gets a reference to the maximum engineering unit value.</summary>
*)
{attribute 'monitoring' := 'call'}
PROPERTY FINAL MaxAnalogValue : REFERENCE TO LREAL
GET
MaxAnalogValue REF= _MaxAnalogValue;
END_GET
END_PROPERTY

(*!
<summary>Gets a reference to the maximum raw process value.</summary>
*)
{attribute 'monitoring' := 'call'}
PROPERTY FINAL MaxRawValue : REFERENCE TO RAW_ANALOG_VALUE
GET
MaxRawValue REF= _MaxRawValue;
END_GET
END_PROPERTY

(*!
<summary>Gets a reference to the minimum engineering unit value.</summary>
*)
{attribute 'monitoring' := 'call'}
PROPERTY FINAL MinAnalogValue : REFERENCE TO LREAL
GET
MinAnalogValue REF= _MinAnalogValue;
END_GET
END_PROPERTY

(*!
<summary>Gets a reference to the minimum raw process value.</summary>
*)
{attribute 'monitoring' := 'call'}
PROPERTY FINAL MinRawValue : REFERENCE TO RAW_ANALOG_VALUE
GET
MinRawValue REF= _MinRawValue;
END_GET
END_PROPERTY

(*!
<summary>Gets the namespace name of the converter.</summary>
*)
{attribute 'monitoring' := 'call'}
PROPERTY NamespaceName : REFERENCE TO STRING
GET
NamespaceName REF= CurrentNamespace.Name;
END_GET
END_PROPERTY

END_FUNCTION_BLOCK

// ---- Analog/StandardConverters/Range/DynamicRangeAnalogValueConverter.TcPOU
(*
SPDX-FileCopyrightText: Â© 2026 Oleksandr Tiutyk <trofimich@gmail.com>
SPDX-License-Identifier: MIT
License: https://opensource.org/license/mit
*)

(*!
<summary>Range converter with dynamically referenced limit variables that can change at runtime.</summary>
<description>
Safely handles online changes without resetting dynamic references to zero.
</description>
*)

{attribute 'no_explicit_call' := 'do not call this function block directly'}
FUNCTION_BLOCK DynamicRangeAnalogValueConverter EXTENDS AbstractRangeAnalogValueConverter
VAR_STAT
	{attribute 'hide'} 
	_ClassName : STRING := __POUNAME();
END_VAR
VAR
	{attribute 'hide'} 
	_ZeroAnalogValue : LREAL;
	{attribute 'hide'} 
	_ZeroRawValue : RAW_ANALOG_VALUE; 
END_VAR

(*!
<summary>Gets the class name of the converter.</summary>
*)
{attribute 'monitoring' := 'call'}
PROPERTY ClassName : REFERENCE TO STRING
GET
ClassName REF= _ClassName;
END_GET
END_PROPERTY

(*!
<summary>Initializes dynamic limit references.</summary>
<param name="bInitRetains">TRUE: retain variables are initialized.</param>
<param name="bInCopyCode">TRUE: instance copied to copy code (online change).</param>
<param name="minAnalogValue">Reference to minimum engineering unit variable.</param>
<param name="maxAnalogValue">Reference to maximum engineering unit variable.</param>
<param name="minRawValue">Reference to minimum raw process variable.</param>
<param name="maxRawValue">Reference to maximum raw process variable.</param>
*)
METHOD FB_init : BOOL
VAR_INPUT
	bInitRetains : BOOL; // TRUE: the retain variables are initialized (reset warm / reset cold)
	bInCopyCode : BOOL;  // TRUE: the instance will be copied to the copy code afterward (online change)
	minAnalogValue : REFERENCE TO LREAL;
	maxAnalogValue : REFERENCE TO LREAL;
	minRawValue : REFERENCE TO RAW_ANALOG_VALUE;
	maxRawValue : REFERENCE TO RAW_ANALOG_VALUE;
END_VAR
IF NOT bInCopyCode THEN
	IF __ISVALIDREF(minAnalogValue) THEN
		_MinAnalogValue REF= minAnalogValue;
	ELSE	
		_MinAnalogValue REF= _ZeroAnalogValue;
	END_IF

	IF __ISVALIDREF(maxAnalogValue) THEN
		_MaxAnalogValue REF= maxAnalogValue;
	ELSE	
		_MaxAnalogValue REF= _ZeroAnalogValue;
	END_IF
		
	IF __ISVALIDREF(minRawValue) THEN
		_MinRawValue REF= minRawValue;
	ELSE	
		_MinRawValue REF= _ZeroRawValue;
	END_IF 

	IF __ISVALIDREF(maxRawValue) THEN
		_MaxRawValue REF= maxRawValue;
	ELSE	
		_MaxRawValue REF= _ZeroRawValue;
	END_IF
END_IF
END_METHOD

(*!
<summary>Gets the memory size of the instance.</summary>
*)
{attribute 'monitoring' := 'call'}
PROPERTY SelfSize : ULINT
GET
SelfSize := XSIZEOF(THIS^);
END_GET
END_PROPERTY

END_FUNCTION_BLOCK

// ---- Analog/StandardConverters/Range/StaticRangeAnalogValueConverter.TcPOU
(*
SPDX-FileCopyrightText: Â© 2026 Oleksandr Tiutyk <trofimich@gmail.com>
SPDX-License-Identifier: MIT
License: https://opensource.org/license/mit
*)

(*!
<summary>Range converter with static limits passed at construction and stored in internal fields.</summary>
<description>
Safely preserves configured limits across TwinCAT online change cycles by guarding against bInCopyCode zeroing.
</description>
*)

{attribute 'no_explicit_call' := 'do not call this function block directly'}
FUNCTION_BLOCK StaticRangeAnalogValueConverter EXTENDS AbstractRangeAnalogValueConverter
VAR_STAT
	{attribute 'hide'} 
	_ClassName : STRING := __POUNAME();
END_VAR
VAR
	{attribute 'hide'} 
	_MinAnalogValueVariable : LREAL;
	{attribute 'hide'} 
	_MaxAnalogValueVariable : LREAL;
	{attribute 'hide'} 
	_MinRawValueVariable : RAW_ANALOG_VALUE;
	{attribute 'hide'} 
	_MaxRawValueVariable : RAW_ANALOG_VALUE;
END_VAR

(*!
<summary>Gets the class name of the converter.</summary>
*)
{attribute 'monitoring' := 'call'}
PROPERTY ClassName : REFERENCE TO STRING
GET
ClassName REF= _ClassName;
END_GET
END_PROPERTY

(*!
<summary>Initializes static limits and binds internal references.</summary>
<param name="bInitRetains">TRUE: retain variables are initialized.</param>
<param name="bInCopyCode">TRUE: instance copied to copy code (online change).</param>
<param name="minAnalogValue">Minimum engineering unit value.</param>
<param name="maxAnalogValue">Maximum engineering unit value.</param>
<param name="minRawValue">Minimum raw hardware process value.</param>
<param name="maxRawValue">Maximum raw hardware process value.</param>
*)
METHOD FB_init : BOOL
VAR_INPUT
	bInitRetains : BOOL; // TRUE: the retain variables are initialized (reset warm / reset cold)
	bInCopyCode : BOOL;  // TRUE: the instance will be copied to the copy code afterward (online change)
	minAnalogValue : LREAL;
	maxAnalogValue : LREAL;
	minRawValue : RAW_ANALOG_VALUE;
	maxRawValue : RAW_ANALOG_VALUE;
END_VAR
IF NOT bInCopyCode THEN
	_MinAnalogValueVariable := minAnalogValue;
	_MaxAnalogValueVariable := maxAnalogValue;
	_MinRawValueVariable := minRawValue;
	_MaxRawValueVariable := maxRawValue;
END_IF

_MinAnalogValue REF= _MinAnalogValueVariable;
_MaxAnalogValue REF= _MaxAnalogValueVariable;
_MinRawValue REF= _MinRawValueVariable;
_MaxRawValue REF= _MaxRawValueVariable;
END_METHOD

(*!
<summary>Gets the memory size of the instance.</summary>
*)
{attribute 'monitoring' := 'call'}
PROPERTY SelfSize : ULINT
GET
SelfSize := XSIZEOF(THIS^);
END_GET
END_PROPERTY

END_FUNCTION_BLOCK

// ---- Digital/Input/DigitalInput.TcPOU
(*
SPDX-FileCopyrightText: Â© 2026 Oleksandr Tiutyk <trofimich@gmail.com>
SPDX-License-Identifier: MIT
License: https://opensource.org/license/mit
*)

(*!
<summary>Digital input automation component supporting normally-open and normally-closed contacts.</summary>
<description>
Reads raw hardware inputs during the automation input processing phase and tracks edge changes.
</description>
*)

FUNCTION_BLOCK DigitalInput EXTENDS TOF_Automation.InputLeafAutomationComponent
	IMPLEMENTS IDigitalInput, TOF_Core.IIOBindable
VAR_STAT
	{attribute 'hide'} 
	_ClassName : STRING := __POUNAME();
END_VAR
VAR
	{attribute 'hide'} 
	_ContactType : CONTACT_TYPE;
	
	_CurrentValue : BOOL;
	_PreviousValue : BOOL;
	
	_RawValue : REFERENCE TO BOOL;
END_VAR

(*!
<summary>Binds component to a raw boolean process image variable.</summary>
<param name="rawValue">Reference to physical boolean input variable.</param>
*)
METHOD BindToIO
VAR_INPUT
	rawValue : REFERENCE TO BOOL;
END_VAR
_RawValue REF= rawValue;
END_METHOD

(*!
<summary>Gets whether the component is bound to a valid physical IO variable.</summary>
*)
{attribute 'monitoring' := 'call'}
PROPERTY FINAL BoundToIO : BOOL
GET
BoundToIO := __ISVALIDREF(_RawValue);
END_GET
END_PROPERTY

(*!
<summary>Indicates whether the logical Value has changed compared to the previous cycle.</summary>
*)
{attribute 'monitoring' := 'call'}
PROPERTY FINAL Changed : BOOL
GET
Changed := _CurrentValue <> _PreviousValue;
END_GET
END_PROPERTY

(*!
<summary>Gets the class name of the component.</summary>
*)
{attribute 'monitoring' := 'call'}
PROPERTY ClassName : REFERENCE TO STRING
GET
ClassName REF= _ClassName;
END_GET
END_PROPERTY

(*!
<summary>Gets or sets electrical contact configuration.</summary>
*)
{attribute 'monitoring' := 'call'}
PROPERTY FINAL ContactType : CONTACT_TYPE
GET
ContactType := _ContactType;
END_GET
SET
_ContactType := ContactType;
END_SET
END_PROPERTY

(*!
<summary>Gets the namespace name of the component.</summary>
*)
{attribute 'monitoring' := 'call'}
PROPERTY NamespaceName : REFERENCE TO STRING
GET
NamespaceName REF= CurrentNamespace.Name;
END_GET
END_PROPERTY

(*!
<summary>Evaluates current input value according to contact type configuration.</summary>
*)
METHOD PROTECTED OnProcessInput
_PreviousValue := _CurrentValue;

IF __ISVALIDREF(_RawValue) THEN
	IF _ContactType = CONTACT_TYPE.NORMALLY_CLOSED THEN
		_CurrentValue := NOT _RawValue;
	ELSE
		_CurrentValue := _RawValue;
	END_IF
END_IF
END_METHOD

(*!
<summary>Gets the memory size of the instance.</summary>
*)
{attribute 'monitoring' := 'call'}
PROPERTY SelfSize : ULINT
GET
SelfSize := XSIZEOF(THIS^);
END_GET
END_PROPERTY

(*!
<summary>Gets evaluated logical boolean state of the input.</summary>
*)
{attribute 'monitoring' := 'call'}
{attribute 'OPC.UA.DA' := '1'}
{attribute 'OPC.UA.DA.Access' := '1'}
PROPERTY FINAL Value : BOOL
GET
Value := _CurrentValue;
END_GET
END_PROPERTY

END_FUNCTION_BLOCK

// ---- Digital/Output/DigitalOutput.TcPOU
(*
SPDX-FileCopyrightText: Â© 2026 Oleksandr Tiutyk <trofimich@gmail.com>
SPDX-License-Identifier: MIT
License: https://opensource.org/license/mit
*)

(*!
<summary>Digital output automation component supporting normally-open and normally-closed contacts.</summary>
<description>
Writes evaluated boolean states to physical hardware outputs during the automation output processing phase.
</description>
*)

FUNCTION_BLOCK DigitalOutput EXTENDS TOF_Automation.OutputLeafAutomationComponent
	IMPLEMENTS IDigitalOutput, TOF_Core.IIOBindable
VAR_STAT
	{attribute 'hide'} 
	_ClassName : STRING := __POUNAME();
END_VAR
VAR
	{attribute 'hide'} 
	_ContactType : CONTACT_TYPE;

	_CurrentValue : BOOL;
	_PreviousValue : BOOL;

	_RawValue : REFERENCE TO BOOL;
END_VAR

(*!
<summary>Binds component to a raw boolean process image output variable.</summary>
<param name="rawValue">Reference to physical boolean output variable.</param>
*)
METHOD BindToIO
VAR_INPUT
	rawValue : REFERENCE TO BOOL;
END_VAR
_RawValue REF= rawValue;
END_METHOD

(*!
<summary>Gets whether the component is bound to a valid physical IO variable.</summary>
*)
{attribute 'monitoring' := 'call'}
PROPERTY FINAL BoundToIO : BOOL
GET
BoundToIO := __ISVALIDREF(_RawValue);
END_GET
END_PROPERTY

(*!
<summary>Indicates whether the current logical command differs from the last processed command.</summary>
<description>
ProcessOutput() acknowledges the current command even without an I/O binding.
</description>
*)
{attribute 'monitoring' := 'call'}
PROPERTY FINAL Changed : BOOL
GET
Changed := _CurrentValue <> _PreviousValue;
END_GET
END_PROPERTY

(*!
<summary>Gets the class name of the component.</summary>
*)
{attribute 'monitoring' := 'call'}
PROPERTY ClassName : REFERENCE TO STRING
GET
ClassName REF= _ClassName;
END_GET
END_PROPERTY

(*!
<summary>Gets or sets electrical contact configuration.</summary>
*)
{attribute 'monitoring' := 'call'}
PROPERTY FINAL ContactType : CONTACT_TYPE
GET
ContactType := _ContactType;
END_GET
SET
_ContactType := ContactType;
END_SET
END_PROPERTY

(*!
<summary>Gets the namespace name of the component.</summary>
*)
{attribute 'monitoring' := 'call'}
PROPERTY NamespaceName : REFERENCE TO STRING
GET
NamespaceName REF= CurrentNamespace.Name;
END_GET
END_PROPERTY

(*!
<summary>Writes logical value to the physical output with contact inversion if configured.</summary>
*)
METHOD PROTECTED OnProcessOutput
IF __ISVALIDREF(_RawValue) THEN
	IF _ContactType = CONTACT_TYPE.NORMALLY_CLOSED THEN
		_RawValue := NOT _CurrentValue;
	ELSE
		_RawValue := _CurrentValue;
	END_IF
END_IF

_PreviousValue := _CurrentValue;
END_METHOD

(*!
<summary>Gets the memory size of the instance.</summary>
*)
{attribute 'monitoring' := 'call'}
PROPERTY SelfSize : ULINT
GET
SelfSize := XSIZEOF(THIS^);
END_GET
END_PROPERTY

(*!
<summary>Gets or sets logical boolean state of the output.</summary>
*)
{attribute 'monitoring' := 'call'}
PROPERTY FINAL Value : BOOL
GET
Value := _CurrentValue;
END_GET
SET
_CurrentValue := Value;
END_SET
END_PROPERTY

END_FUNCTION_BLOCK
